// TIA Portal V16 export
// export: Created 2024-09-05T17:39:14.1458519Z, ExportSetting WithDefaults, DisplayName Totally Integrated Automation Portal, DisplayVersion V16 Update 6, DisplayName TIA Portal Version Control Interface, DisplayVersion V16 Update 2, DisplayName TIA Portal Openness, DisplayVersion V16 Update 6, DisplayName STEP 7 Professional, DisplayVersion V16 Update 6, DisplayName STEP 7 Safety, DisplayVersion V16, DisplayName WinCC Advanced, DisplayVersion V16 Update 6
DATA_BLOCK "Cylinders_Commands"   // DB12
{ S7_Optimized_Access := 'FALSE' }
VERSION : 0.1
// stored: AutoNumber false, DBAccessibleFromOPCUA true, IsOnlyStoredInLoadMemory false, IsWriteProtectedInAS false
   VAR RETAIN
      VH1 { S7_SetPoint := 'True'} : "UDT_HydraulicCylinderData";
      VH2 { S7_SetPoint := 'True'} : "UDT_HydraulicCylinderData";
      VH3 { S7_SetPoint := 'True'} : "UDT_HydraulicCylinderData";
      VH4 { S7_SetPoint := 'True'} : "UDT_HydraulicCylinderData";
   END_VAR
BEGIN
   VH1.Pressure := 0.0;
   VH1.Flow := 0.0;
   VH1.Position := 0.0;
   VH1.StandstillPosition := 0.0;
   VH1.PressureCmd := 0.0;
   VH1.FlowCmd := 0.0;
   VH1.PressureBack := 0.0;
   VH1.FlowBack := 0.0;
   VH1.HAxis := 0.0;
   VH1.Force := 0.0;
   VH1.Status.InWp := FALSE;
   VH1.Status.InBp := FALSE;
   VH1.Status.InFp := FALSE;
   VH1.Status.ToWp := FALSE;
   VH1.Status.ToBp := FALSE;
   VH1.Status.ToFp := FALSE;
   VH1.InBp_1mm_margin := FALSE;
   VH2.Pressure := 0.0;
   VH2.Flow := 0.0;
   VH2.Position := 0.0;
   VH2.StandstillPosition := 0.0;
   VH2.PressureCmd := 0.0;
   VH2.FlowCmd := 0.0;
   VH2.PressureBack := 0.0;
   VH2.FlowBack := 0.0;
   VH2.HAxis := 0.0;
   VH2.Force := 0.0;
   VH2.Status.InWp := FALSE;
   VH2.Status.InBp := FALSE;
   VH2.Status.InFp := FALSE;
   VH2.Status.ToWp := FALSE;
   VH2.Status.ToBp := FALSE;
   VH2.Status.ToFp := FALSE;
   VH2.InBp_1mm_margin := FALSE;
   VH3.Pressure := 0.0;
   VH3.Flow := 0.0;
   VH3.Position := 5.820313;
   VH3.StandstillPosition := 0.0;
   VH3.PressureCmd := 0.0;
   VH3.FlowCmd := 0.0;
   VH3.PressureBack := 0.0;
   VH3.FlowBack := 0.0;
   VH3.HAxis := 0.0;
   VH3.Force := 0.0;
   VH3.Status.InWp := FALSE;
   VH3.Status.InBp := FALSE;
   VH3.Status.InFp := FALSE;
   VH3.Status.ToWp := FALSE;
   VH3.Status.ToBp := FALSE;
   VH3.Status.ToFp := FALSE;
   VH3.InBp_1mm_margin := FALSE;
   VH4.Pressure := 0.0;
   VH4.Flow := 0.0;
   VH4.Position := 4.661458;
   VH4.StandstillPosition := 0.0;
   VH4.PressureCmd := 0.0;
   VH4.FlowCmd := 0.0;
   VH4.PressureBack := 0.0;
   VH4.FlowBack := 0.0;
   VH4.HAxis := 0.0;
   VH4.Force := 0.0;
   VH4.Status.InWp := FALSE;
   VH4.Status.InBp := FALSE;
   VH4.Status.InFp := FALSE;
   VH4.Status.ToWp := FALSE;
   VH4.Status.ToBp := FALSE;
   VH4.Status.ToFp := FALSE;
   VH4.InBp_1mm_margin := FALSE;
END_DATA_BLOCK
